PROGRAM MAIN
VAR
	wText : 'Hello world';
	
END_VAR

END_PROGRAM

(* stored: Version 1.1.0.1, ProductVersion 3.1.4024.9
   POU MAIN: Id {d0e89976-a164-4fff-a0bc-f3c1f106537c}, SpecialFunc None *)
